// TIA Portal V19 export
FUNCTION_BLOCK "Decoiler_FB"   // FB72, LAD
TITLE = DECOILER MOUNTED ON A ROTATION SYSTEM FOR ON-LINE/OFF-LINE EXCHANGE
// stored: MemoryReserve 100, SetENOAutomatically false
   VAR_INPUT
      AreaInterface : "AreaInterface";
      ZSI : "udt_ZoneSafetyInterface";
      DSI : Struct
         Feed : "udt_DeviceSafetyInterface";
         Jaws : "udt_DeviceSafetyInterface";
         Coupling : "udt_DeviceSafetyInterface";
         SnubberLift : "udt_DeviceSafetyInterface";
         SnubberRoll : "udt_DeviceSafetyInterface";
      END_STRUCT;
      Drive : "TAx_DriveInterface";
      HW_ID_TEL1 : HW_SUBMODULE;
      DataIn : Struct
         DiameterSensor : Int;
         LsPosizioneRazza : Bool;
         Feed : "SpeedMachine_DataIn";
         Jaws : "ValveMachine_DataIn";
         Coupling : "ValveMachine_DataIn";
         SnubberLift : "ValveMachine_DataIn";
         SnubberRoll : "ValveMachine_DataIn";
         Loop : Struct
            Connector : Bool;
            S_MinHigh : Bool;
            S_SpeedAsjust : Bool;
            S_MaxLow : Bool;
         END_STRUCT;
         PneumaticBrake : Struct
            PbOpenClose : Bool;
            PbPartialOpenClose : Bool;
         END_STRUCT;
      END_STRUCT;
      CIn : Struct
         Manager : "Decoiler_Manager";
         PressureRunning : Bool;
      END_STRUCT;
      Config : Struct
         Loop : Struct
            Exist_S_MinHigh : Bool;
            Exist_S_SpeedAdjust : Bool;
         END_STRUCT;
         Feed : "SpeedMachine_Config";
         Jaws : "ValveMachine_Config";
         Coupling : "ValveMachine_Config";
         SnubberLift : "ValveMachine_Config";
         SnubberRoll : "ValveMachine_Config";
         Enable_End_Of_Coil_Using_Loop : Bool := FALSE;
      END_STRUCT;
   END_VAR
   VAR_OUTPUT
      MachineInterface : "MachineInterface";
      DataOut : Struct
         Feed : "SpeedMachine_DataOut";
         Jaws : "ValveMachine_DataOut";
         Coupling : "ValveMachine_DataOut";
         SnubberLift : "ValveMachine_DataOut";
         SnubberRoll : "ValveMachine_DataOut";
         PneumaticBrake : Struct
            V_Open : Bool;
            V_PartialHigh : Bool;
            V_PartialLow : Bool;
            Lp_PbPartialBrake : Bool;
         END_STRUCT;
      END_STRUCT;
      COut : "Decoiler_Status";
   END_VAR
   VAR_IN_OUT
      PersistentValues : "Decoiler_Pers";
   END_VAR
   VAR
      Alarm : Struct
         Feed : "SpeedMachine_Alr";
         Jaws : "ValveAlr";
         Coupling : "ValveAlr";
         SnubberLift : "ValveAlr";
         SnubberRoll : "ValveAlr";
         DimeterSensor : Struct
            SensorrPresetNeed { ExternalAccessible := 'False'; ExternalVisible := 'False'; ExternalWritable := 'False'} : Bool;
         END_STRUCT;
         Loop : Struct
            ConnectorUnplugged : Bool;
         END_STRUCT;
      END_STRUCT;
      Warning : Struct
         EndCoilDetect : Bool;
         Feed : "SpeedMachine_Wng";
         Jaws : "ValveMachine_Wng";
         Coupling { S7_SetPoint := 'True'} : "ValveMachine_Wng";
         SnubberLift { S7_SetPoint := 'True'} : "ValveMachine_Wng";
         SnubberRoll { S7_SetPoint := 'True'} : "ValveMachine_Wng";
         Loop : Struct
            MinHigh : Bool;
         END_STRUCT;
      END_STRUCT;
      HMI : Struct
         Diameter_ButtonPreset : Bool;
         Diameter_PresetValue : Real;
      END_STRUCT;
      Sts : Struct
         StopPosizioneRazza : Bool;
      END_STRUCT;
      Ctrl : Struct
         Jaws : Struct
            AutoOpen : Bool;
            TON_Pause : IEC_TIMER;
            TON_Duration : IEC_TIMER;
         END_STRUCT;
         Brake : Struct
            Open_ReqByMotor : Bool;
            TON_PartialOFF : IEC_TIMER;
            TON_OpenOFF : IEC_TIMER;
         END_STRUCT;
      END_STRUCT;
      DiameterSensor { S7_SetPoint := 'True'} : "Decoiler_DiameterSensor_FB";
      Loop { S7_SetPoint := 'True'} : "Decoiler_Loop_FB";
      Feed { S7_SetPoint := 'True'} : "SpeedMachine_FB";
      PneumaticBrake { S7_SetPoint := 'True'} : "Decoiler_PneumaticBrake";
      Jaws { S7_SetPoint := 'True'} : "ValveMachine_FB";
      SnubberLift { S7_SetPoint := 'True'} : "ValveMachine_FB";
      SnubberRoll { S7_SetPoint := 'True'} : "ValveMachine_FB";
      Coupling { S7_SetPoint := 'True'} : "ValveMachine_FB";
      TON_EndCoilDetect : IEC_TIMER;
      AuxPE : Struct
         LsPosizioneRazza : Bool;
      END_STRUCT;
   END_VAR
   VAR_TEMP
      PE : Struct
         LsPosizioneRazza : Bool;
      END_STRUCT;
      Req : Bool;
   END_VAR
   VAR CONSTANT
      PI : LReal := 3.14159265358979;
   END_VAR
   VAR_TEMP   // added for the SCL form of the ladder/FBD networks
      _w1 : Bool;
   END_VAR
BEGIN

REGION Network 1: <<< MATERIAL FEEDING - PAY-OFF BKW / FWD >>>
END_REGION

REGION Network 2: < Coil Diameter >
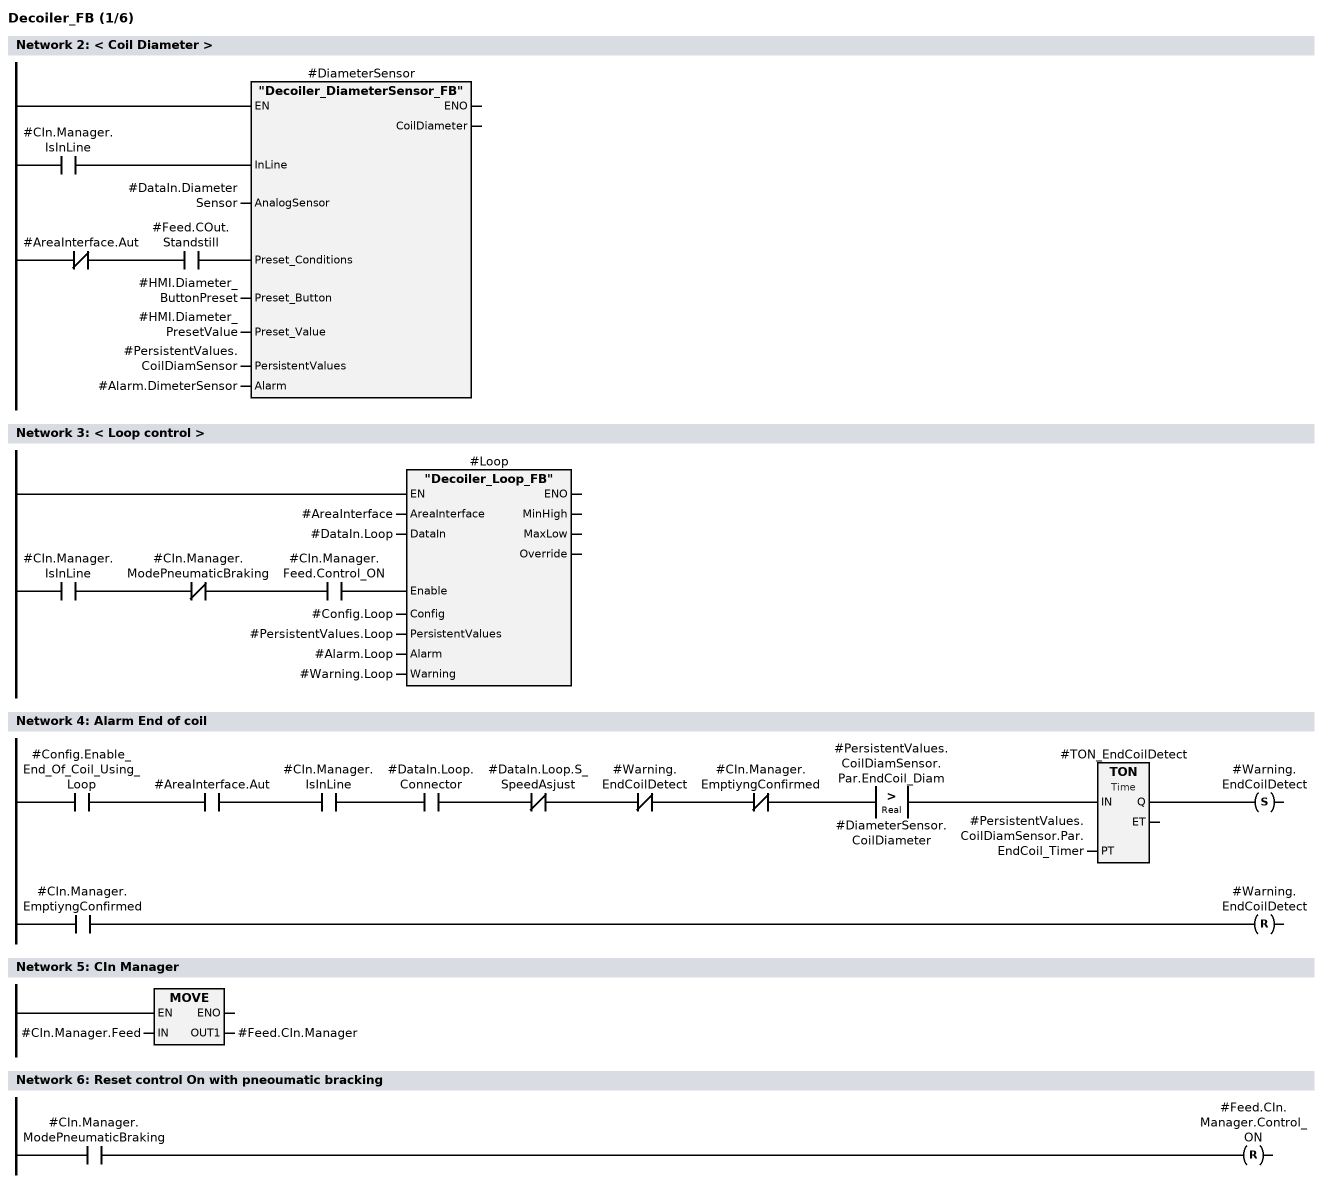
   RUNG wire#powerrail
      #DiameterSensor(InLine := wire#w1, Preset_Conditions := wire#w2, AnalogSensor := #DataIn.DiameterSensor, Preset_Button := #HMI.Diameter_ButtonPreset, Preset_Value := #HMI.Diameter_PresetValue, PersistentValues := #PersistentValues.CoilDiamSensor, Alarm := #Alarm.DimeterSensor, CoilDiameter =>)
   END_RUNG
   RUNG wire#powerrail
      Contact( #CIn.Manager.IsInLine )
   END_RUNG wire#w1
   RUNG wire#powerrail
      I_Contact( #AreaInterface.Aut )
      Contact( #Feed.COut.Standstill )
   END_RUNG wire#w2
   // the same network as SCL:
   #DiameterSensor(InLine := #CIn.Manager.IsInLine,   // "Decoiler_DiameterSensor_FB"
                   AnalogSensor := #DataIn.DiameterSensor,
                   Preset_Conditions := NOT #AreaInterface.Aut AND #Feed.COut.Standstill,
                   Preset_Button := #HMI.Diameter_ButtonPreset,
                   Preset_Value := #HMI.Diameter_PresetValue,
                   PersistentValues := #PersistentValues.CoilDiamSensor,
                   Alarm := #Alarm.DimeterSensor);
END_REGION

REGION Network 3: < Loop control >
   RUNG wire#powerrail
      #Loop(Enable := wire#w1, AreaInterface := #AreaInterface, DataIn := #DataIn.Loop, Config := #Config.Loop, PersistentValues := #PersistentValues.Loop, Alarm := #Alarm.Loop, Warning := #Warning.Loop, MinHigh =>, MaxLow =>, Override =>)
   END_RUNG
   RUNG wire#powerrail
      Contact( #CIn.Manager.IsInLine )
      I_Contact( #CIn.Manager.ModePneumaticBraking )
      Contact( #CIn.Manager.Feed.Control_ON )
   END_RUNG wire#w1
   // the same network as SCL:
   #Loop(AreaInterface := #AreaInterface,   // "Decoiler_Loop_FB"
         DataIn := #DataIn.Loop,
         Enable := #CIn.Manager.IsInLine AND NOT #CIn.Manager.ModePneumaticBraking AND #CIn.Manager.Feed.Control_ON,
         Config := #Config.Loop,
         PersistentValues := #PersistentValues.Loop,
         Alarm := #Alarm.Loop,
         Warning := #Warning.Loop);
END_REGION

REGION Network 4: Alarm End of coil
   RUNG wire#powerrail
      Contact( #Config.Enable_End_Of_Coil_Using_Loop )
      Contact( #AreaInterface.Aut )
      Contact( #CIn.Manager.IsInLine )
      Contact( #DataIn.Loop.Connector )
      I_Contact( #DataIn.Loop.S_SpeedAsjust )
      I_Contact( #Warning.EndCoilDetect )
      I_Contact( #CIn.Manager.EmptiyngConfirmed )
      { S7_Templates := "SrcType := Real" } GT_Contact(in1 := #PersistentValues.CoilDiamSensor.Par.EndCoil_Diam, in2 := #DiameterSensor.CoilDiameter)
      { S7_Templates := "time_type := Time" } #TON_EndCoilDetect.TON(pt := #PersistentValues.CoilDiamSensor.Par.EndCoil_Timer, et =>)
      S_Coil( #Warning.EndCoilDetect )
   END_RUNG
   RUNG wire#powerrail
      Contact( #CIn.Manager.EmptiyngConfirmed )
      R_Coil( #Warning.EndCoilDetect )
   END_RUNG
   // the same network as SCL:
   #TON_EndCoilDetect.TON(IN := #Config.Enable_End_Of_Coil_Using_Loop AND #AreaInterface.Aut AND #CIn.Manager.IsInLine AND #DataIn.Loop.Connector AND NOT #DataIn.Loop.S_SpeedAsjust AND NOT #Warning.EndCoilDetect AND NOT #CIn.Manager.EmptiyngConfirmed AND (#PersistentValues.CoilDiamSensor.Par.EndCoil_Diam > #DiameterSensor.CoilDiameter),
                          PT := #PersistentValues.CoilDiamSensor.Par.EndCoil_Timer);
   IF #TON_EndCoilDetect.Q THEN #Warning.EndCoilDetect := TRUE; END_IF;
   IF #CIn.Manager.EmptiyngConfirmed THEN #Warning.EndCoilDetect := FALSE; END_IF;
END_REGION

REGION Network 5: CIn Manager
   RUNG wire#powerrail
      Move(in := #CIn.Manager.Feed, out1 => #Feed.CIn.Manager)
   END_RUNG
   // the same network as SCL:
   #Feed.CIn.Manager := #CIn.Manager.Feed;
END_REGION

REGION Network 6: Reset control On with pneoumatic bracking
   RUNG wire#powerrail
      Contact( #CIn.Manager.ModePneumaticBraking )
      R_Coil( #Feed.CIn.Manager.Control_ON )
   END_RUNG
   // the same network as SCL:
   IF #CIn.Manager.ModePneumaticBraking THEN #Feed.CIn.Manager.Control_ON := FALSE; END_IF;
END_REGION

REGION Network 7 (SCL): Velocity override with no coupling

   IF NOT #PersistentValues.Coupling.Engaged OR
       NOT #Coupling.COut.Work
   THEN
       #Feed.CIn.Manager.Vel := #PersistentValues.Feed.Man.VelFwdHigh;
   END_IF;
END_REGION

REGION Network 8: CIn Velocity Override
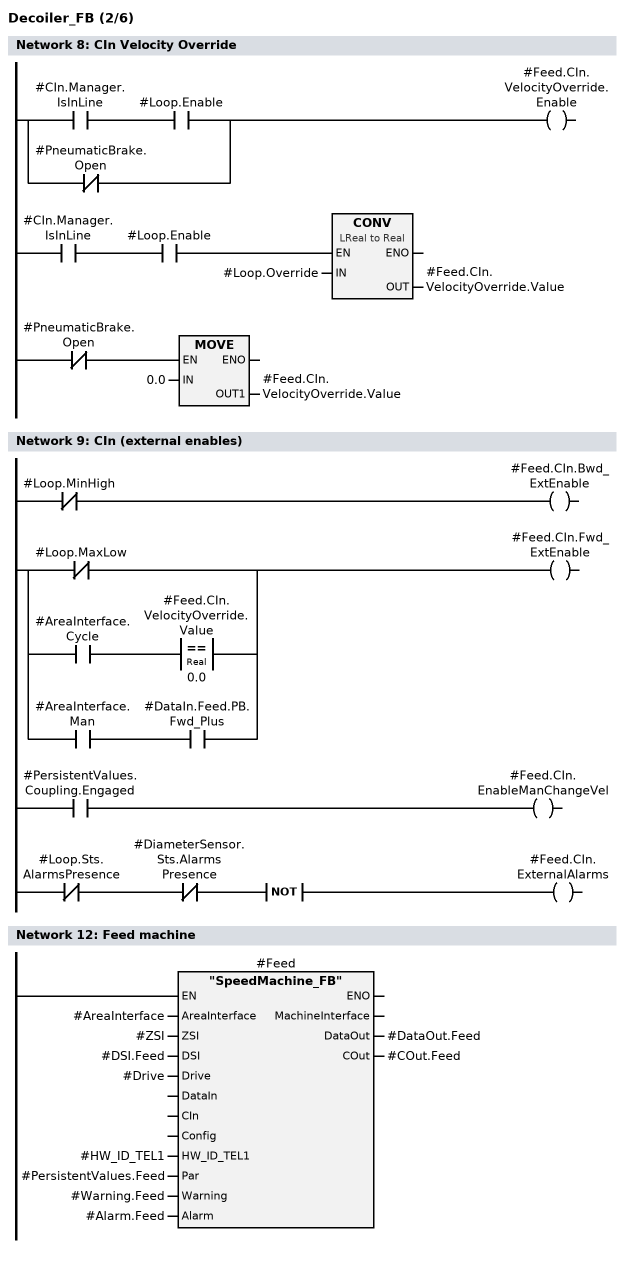
   RUNG wire#powerrail
      Contact( #CIn.Manager.IsInLine )
      Contact( #Loop.Enable )
      wire#w1
      Coil( #Feed.CIn.VelocityOverride.Enable )
   END_RUNG
   RUNG wire#powerrail
      I_Contact( #PneumaticBrake.Open )
   END_RUNG wire#w1
   RUNG wire#powerrail
      Contact( #CIn.Manager.IsInLine )
      Contact( #Loop.Enable )
      { S7_Templates := "[SrcType := LReal, DestType := Real]" } Convert(in := #Loop.Override, out => #Feed.CIn.VelocityOverride.Value)
   END_RUNG
   RUNG wire#powerrail
      I_Contact( #PneumaticBrake.Open )
      Move(in := 0.0, out1 => #Feed.CIn.VelocityOverride.Value)
   END_RUNG
   // the same network as SCL:
   #Feed.CIn.VelocityOverride.Enable := (#CIn.Manager.IsInLine AND #Loop.Enable) OR NOT #PneumaticBrake.Open;
   IF #CIn.Manager.IsInLine AND #Loop.Enable THEN
       #Feed.CIn.VelocityOverride.Value := LREAL_TO_REAL(#Loop.Override);
   END_IF;
   IF NOT #PneumaticBrake.Open THEN #Feed.CIn.VelocityOverride.Value := 0.0; END_IF;
END_REGION

REGION Network 9: CIn (external enables)
   RUNG wire#powerrail
      I_Contact( #Loop.MinHigh )
      Coil( #Feed.CIn.Bwd_ExtEnable )
   END_RUNG
   RUNG wire#powerrail
      I_Contact( #Loop.MaxLow )
      wire#w1
      Coil( #Feed.CIn.Fwd_ExtEnable )
   END_RUNG
   RUNG wire#powerrail
      Contact( #AreaInterface.Cycle )
      { S7_Templates := "SrcType := Real" } EQ_Contact(in1 := #Feed.CIn.VelocityOverride.Value, in2 := 0.0)
   END_RUNG wire#w1
   RUNG wire#powerrail
      Contact( #AreaInterface.Man )
      Contact( #DataIn.Feed.PB.Fwd_Plus )
   END_RUNG wire#w1
   RUNG wire#powerrail
      Contact( #PersistentValues.Coupling.Engaged )
      Coil( #Feed.CIn.EnableManChangeVel )
   END_RUNG
   RUNG wire#powerrail
      I_Contact( #Loop.Sts.AlarmsPresence )
      I_Contact( #DiameterSensor.Sts.AlarmsPresence )
      Not()
      Coil( #Feed.CIn.ExternalAlarms )
   END_RUNG
   // the same network as SCL:
   #Feed.CIn.Bwd_ExtEnable := NOT #Loop.MinHigh;
   #Feed.CIn.Fwd_ExtEnable := NOT #Loop.MaxLow OR (#AreaInterface.Cycle AND (#Feed.CIn.VelocityOverride.Value = 0.0)) OR (#AreaInterface.Man AND #DataIn.Feed.PB.Fwd_Plus);
   #Feed.CIn.EnableManChangeVel := #PersistentValues.Coupling.Engaged;
   #Feed.CIn.ExternalAlarms := NOT (NOT #Loop.Sts.AlarmsPresence AND NOT #DiameterSensor.Sts.AlarmsPresence);
END_REGION

REGION Network 10 (SCL): Config
   #Feed.Config := #Config.Feed;


   #Feed.Config.Ax.LeadScrewPitchVal := #PI * #DiameterSensor.CoilDiameter;
END_REGION

REGION Network 11 (SCL): Data In
   #Feed.DataIn := #DataIn.Feed;

   #PE.LsPosizioneRazza := #DataIn.LsPosizioneRazza AND NOT #AuxPE.LsPosizioneRazza;
   #AuxPE.LsPosizioneRazza := #DataIn.LsPosizioneRazza;

   IF (#DataIn.Feed.PB.Fwd_Plus OR #DataIn.Feed.PB.Bwd_Minus) AND
       #PE.LsPosizioneRazza
   THEN
       #Sts.StopPosizioneRazza := TRUE;
   ELSIF NOT #DataIn.Feed.PB.Fwd_Plus AND
       NOT #DataIn.Feed.PB.Bwd_Minus
   THEN
       #Sts.StopPosizioneRazza := FALSE;
   END_IF;

   #Feed.DataIn.PB.Fwd_Plus := #DataIn.Feed.PB.Fwd_Plus AND NOT #Sts.StopPosizioneRazza;
   #Feed.DataIn.PB.Bwd_Minus := #DataIn.Feed.PB.Bwd_Minus AND NOT #Sts.StopPosizioneRazza;
END_REGION

REGION Network 12: Feed machine
   RUNG wire#powerrail
      #Feed(AreaInterface := #AreaInterface, ZSI := #ZSI, DSI := #DSI.Feed, Drive := #Drive, DataIn :=, CIn :=, Config :=, HW_ID_TEL1 := #HW_ID_TEL1, Par := #PersistentValues.Feed, Warning := #Warning.Feed, Alarm := #Alarm.Feed, MachineInterface =>, DataOut => #DataOut.Feed, COut => #COut.Feed)
   END_RUNG
   // the same network as SCL:
   #Feed(AreaInterface := #AreaInterface,   // "SpeedMachine_FB"
         ZSI := #ZSI,
         DSI := #DSI.Feed,
         Drive := #Drive,
         HW_ID_TEL1 := #HW_ID_TEL1,
         Par := #PersistentValues.Feed,
         Warning := #Warning.Feed,
         Alarm := #Alarm.Feed,
         DataOut => #DataOut.Feed,
         COut => #COut.Feed);
END_REGION

REGION Network 13: < Pneumatic brake >
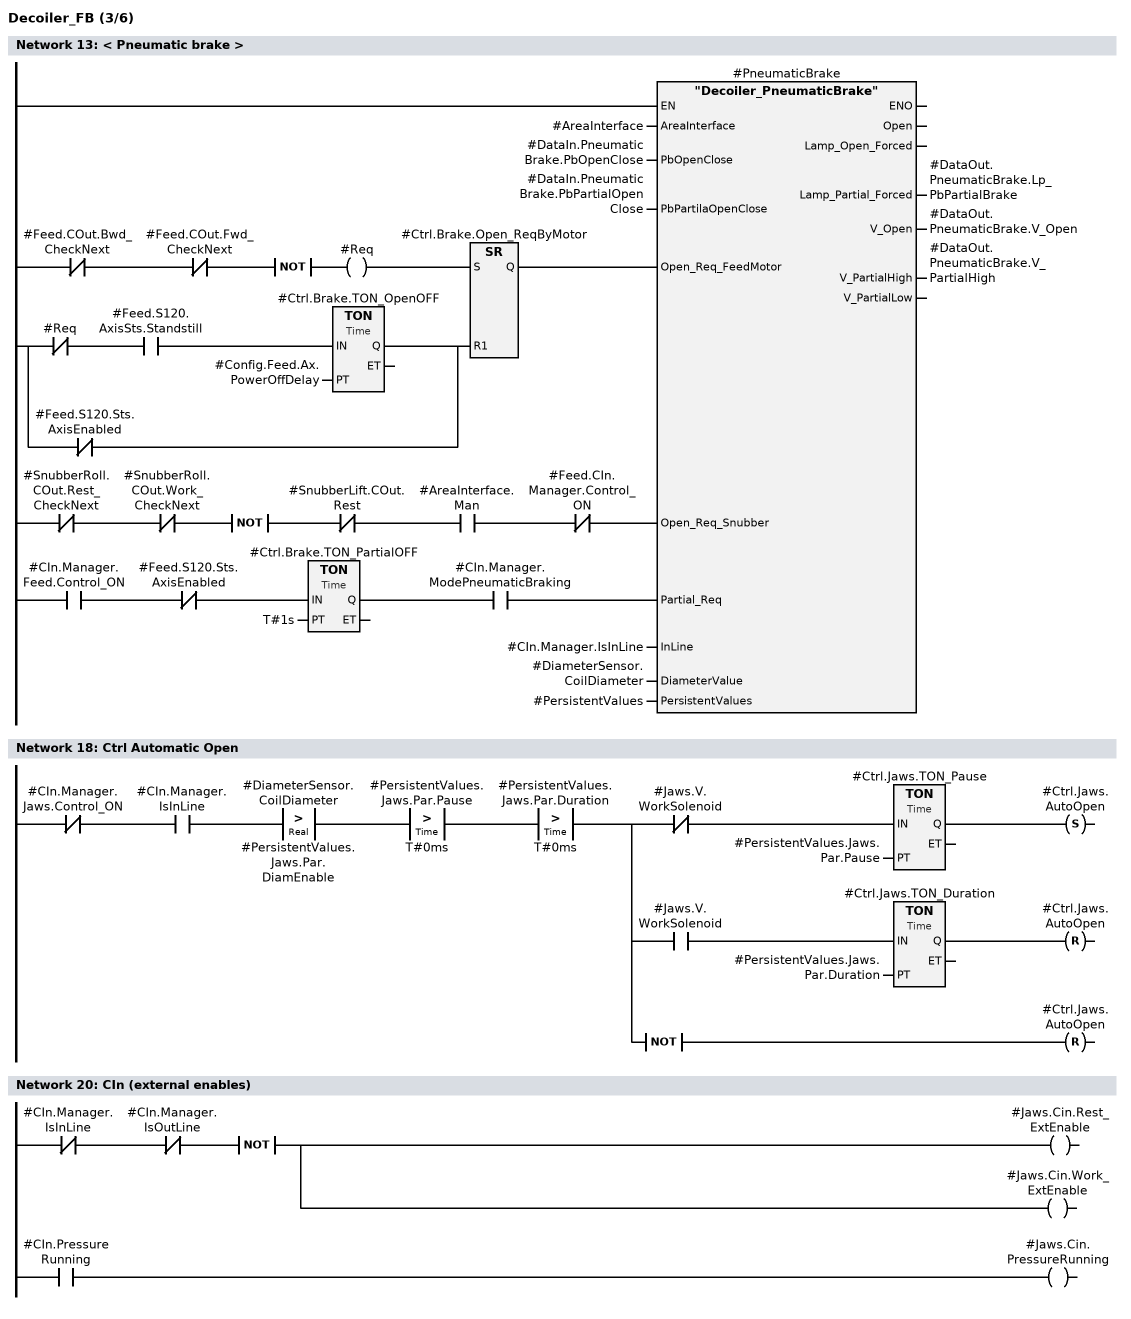
   RUNG wire#powerrail
      #PneumaticBrake(Open_Req_FeedMotor := wire#w2, Open_Req_Snubber := wire#w3, Partial_Req := wire#w4, AreaInterface := #AreaInterface, PbOpenClose := #DataIn.PneumaticBrake.PbOpenClose, PbPartilaOpenClose := #DataIn.PneumaticBrake.PbPartialOpenClose, InLine := #CIn.Manager.IsInLine, DiameterValue := #DiameterSensor.CoilDiameter, PersistentValues := #PersistentValues, Open =>, Lamp_Open_Forced =>, Lamp_Partial_Forced => #DataOut.PneumaticBrake.Lp_PbPartialBrake, V_Open => #DataOut.PneumaticBrake.V_Open, V_PartialHigh => #DataOut.PneumaticBrake.V_PartialHigh, V_PartialLow =>)
   END_RUNG
   RUNG wire#powerrail
      I_Contact( #Feed.COut.Bwd_CheckNext )
      I_Contact( #Feed.COut.Fwd_CheckNext )
      Not()
      Coil( #Req )
      S_SR(operand := #Ctrl.Brake.Open_ReqByMotor, r1 := wire#w1)
   END_RUNG wire#w2
   RUNG wire#powerrail
      I_Contact( #Req )
      Contact( #Feed.S120.AxisSts.Standstill )
      { S7_Templates := "time_type := Time" } #Ctrl.Brake.TON_OpenOFF.TON(pt := #Config.Feed.Ax.PowerOffDelay, et =>)
   END_RUNG wire#w1
   RUNG wire#powerrail
      I_Contact( #Feed.S120.Sts.AxisEnabled )
   END_RUNG wire#w1
   RUNG wire#powerrail
      I_Contact( #SnubberRoll.COut.Rest_CheckNext )
      I_Contact( #SnubberRoll.COut.Work_CheckNext )
      Not()
      I_Contact( #SnubberLift.COut.Rest )
      Contact( #AreaInterface.Man )
      I_Contact( #Feed.CIn.Manager.Control_ON )
   END_RUNG wire#w3
   RUNG wire#powerrail
      Contact( #CIn.Manager.Feed.Control_ON )
      I_Contact( #Feed.S120.Sts.AxisEnabled )
      { S7_Templates := "time_type := Time" } #Ctrl.Brake.TON_PartialOFF.TON(pt := T#1s, et =>)
      Contact( #CIn.Manager.ModePneumaticBraking )
   END_RUNG wire#w4
   // the same network as SCL:
   #Req := NOT (NOT #Feed.COut.Bwd_CheckNext AND NOT #Feed.COut.Fwd_CheckNext);
   #Ctrl.Brake.TON_OpenOFF.TON(IN := NOT #Req AND #Feed.S120.AxisSts.Standstill,
                           PT := #Config.Feed.Ax.PowerOffDelay);
   IF #Req THEN
       #Ctrl.Brake.Open_ReqByMotor := TRUE;   // SR flip-flop
   END_IF;
   IF #Ctrl.Brake.TON_OpenOFF.Q OR NOT #Feed.S120.Sts.AxisEnabled THEN
       #Ctrl.Brake.Open_ReqByMotor := FALSE;
   END_IF;
   #Ctrl.Brake.TON_PartialOFF.TON(IN := #CIn.Manager.Feed.Control_ON AND NOT #Feed.S120.Sts.AxisEnabled,
                           PT := T#1s);
   #PneumaticBrake(AreaInterface := #AreaInterface,   // "Decoiler_PneumaticBrake"
                   PbOpenClose := #DataIn.PneumaticBrake.PbOpenClose,
                   PbPartilaOpenClose := #DataIn.PneumaticBrake.PbPartialOpenClose,
                   Open_Req_FeedMotor := #Ctrl.Brake.Open_ReqByMotor,
                   Open_Req_Snubber := NOT (NOT #SnubberRoll.COut.Rest_CheckNext AND NOT #SnubberRoll.COut.Work_CheckNext) AND NOT #SnubberLift.COut.Rest AND #AreaInterface.Man AND NOT #Feed.CIn.Manager.Control_ON,
                   Partial_Req := #Ctrl.Brake.TON_PartialOFF.Q AND #CIn.Manager.ModePneumaticBraking,
                   InLine := #CIn.Manager.IsInLine,
                   DiameterValue := #DiameterSensor.CoilDiameter,
                   PersistentValues := #PersistentValues,
                   Lamp_Partial_Forced => #DataOut.PneumaticBrake.Lp_PbPartialBrake,
                   V_Open => #DataOut.PneumaticBrake.V_Open,
                   V_PartialHigh => #DataOut.PneumaticBrake.V_PartialHigh);
END_REGION

REGION Network 14: >
END_REGION

REGION Network 15: >
END_REGION

REGION Network 16: >
END_REGION

REGION Network 17: <<< JAWS CLOSE / OPEN >>>
END_REGION

REGION Network 18: Ctrl Automatic Open
   RUNG wire#powerrail
      I_Contact( #CIn.Manager.Jaws.Control_ON )
      Contact( #CIn.Manager.IsInLine )
      { S7_Templates := "SrcType := Real" } GT_Contact(in1 := #DiameterSensor.CoilDiameter, in2 := #PersistentValues.Jaws.Par.DiamEnable)
      { S7_Templates := "SrcType := Time" } GT_Contact(in1 := #PersistentValues.Jaws.Par.Pause, in2 := T#0ms)
      { S7_Templates := "SrcType := Time" } GT_Contact(in1 := #PersistentValues.Jaws.Par.Duration, in2 := T#0ms)
      wire#w1
      I_Contact( #Jaws.V.WorkSolenoid )
      { S7_Templates := "time_type := Time" } #Ctrl.Jaws.TON_Pause.TON(pt := #PersistentValues.Jaws.Par.Pause, et =>)
      S_Coil( #Ctrl.Jaws.AutoOpen )
   END_RUNG
   RUNG wire#w1
      Contact( #Jaws.V.WorkSolenoid )
      { S7_Templates := "time_type := Time" } #Ctrl.Jaws.TON_Duration.TON(pt := #PersistentValues.Jaws.Par.Duration, et =>)
      R_Coil( #Ctrl.Jaws.AutoOpen )
   END_RUNG
   RUNG wire#w1
      Not()
      R_Coil( #Ctrl.Jaws.AutoOpen )
   END_RUNG
   // the same network as SCL:
   #_w1 := NOT #CIn.Manager.Jaws.Control_ON AND #CIn.Manager.IsInLine AND (#DiameterSensor.CoilDiameter > #PersistentValues.Jaws.Par.DiamEnable) AND (#PersistentValues.Jaws.Par.Pause > T#0ms) AND (#PersistentValues.Jaws.Par.Duration > T#0ms);
   #Ctrl.Jaws.TON_Pause.TON(IN := #_w1 AND NOT #Jaws.V.WorkSolenoid, PT := #PersistentValues.Jaws.Par.Pause);
   IF #Ctrl.Jaws.TON_Pause.Q THEN #Ctrl.Jaws.AutoOpen := TRUE; END_IF;
   #Ctrl.Jaws.TON_Duration.TON(IN := #_w1 AND #Jaws.V.WorkSolenoid, PT := #PersistentValues.Jaws.Par.Duration);
   IF #Ctrl.Jaws.TON_Duration.Q THEN #Ctrl.Jaws.AutoOpen := FALSE; END_IF;
   IF NOT #_w1 THEN #Ctrl.Jaws.AutoOpen := FALSE; END_IF;
END_REGION

REGION Network 19 (SCL): CIn Manager
   #Jaws.Cin.Manager := #CIn.Manager.Jaws;

   IF NOT #CIn.Manager.Jaws.Control_ON AND #CIn.Manager.IsInLine THEN

       #Jaws.Cin.Manager.Control_ON := #Ctrl.Jaws.AutoOpen;
       #Jaws.Cin.Manager.Work := #Ctrl.Jaws.AutoOpen;
       #Jaws.Cin.Manager.Rest := FALSE;

   END_IF;
END_REGION

REGION Network 20: CIn (external enables)
   RUNG wire#powerrail
      I_Contact( #CIn.Manager.IsInLine )
      I_Contact( #CIn.Manager.IsOutLine )
      Not()
      wire#w1
      Coil( #Jaws.Cin.Rest_ExtEnable )
   END_RUNG
   RUNG wire#w1
      Coil( #Jaws.Cin.Work_ExtEnable )
   END_RUNG
   RUNG wire#powerrail
      Contact( #CIn.PressureRunning )
      Coil( #Jaws.Cin.PressureRunning )
   END_RUNG
   // the same network as SCL:
   #Jaws.Cin.Rest_ExtEnable := NOT (NOT #CIn.Manager.IsInLine AND NOT #CIn.Manager.IsOutLine);
   #Jaws.Cin.Work_ExtEnable := #Jaws.Cin.Rest_ExtEnable;
   #Jaws.Cin.PressureRunning := #CIn.PressureRunning;
END_REGION

REGION Network 21: Valve machine
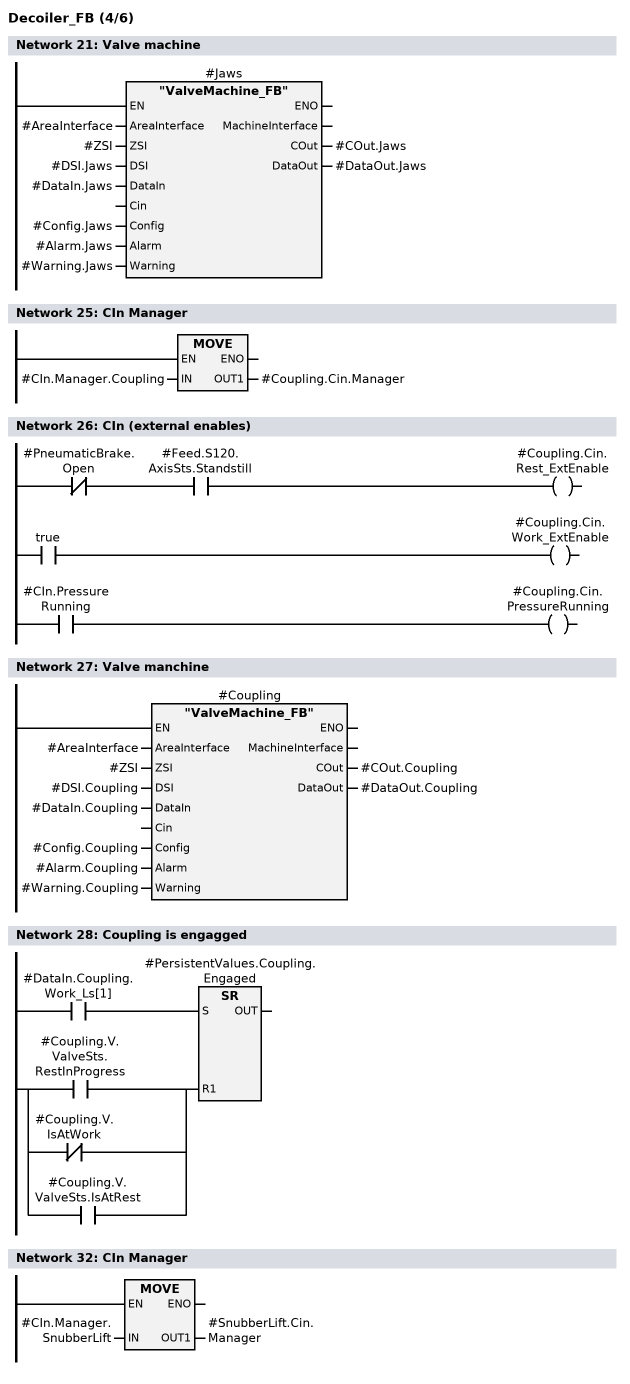
   RUNG wire#powerrail
      #Jaws(AreaInterface := #AreaInterface, ZSI := #ZSI, DSI := #DSI.Jaws, DataIn := #DataIn.Jaws, Cin :=, Config := #Config.Jaws, Alarm := #Alarm.Jaws, Warning := #Warning.Jaws, MachineInterface =>, COut => #COut.Jaws, DataOut => #DataOut.Jaws)
   END_RUNG
   // the same network as SCL:
   #Jaws(AreaInterface := #AreaInterface,   // "ValveMachine_FB"
         ZSI := #ZSI,
         DSI := #DSI.Jaws,
         DataIn := #DataIn.Jaws,
         Config := #Config.Jaws,
         Alarm := #Alarm.Jaws,
         Warning := #Warning.Jaws,
         COut => #COut.Jaws,
         DataOut => #DataOut.Jaws);
END_REGION

REGION Network 22: >
END_REGION

REGION Network 23: >
END_REGION

REGION Network 24: <<< MOTOR COUPLING WORK / REST >>>
END_REGION

REGION Network 25: CIn Manager
   RUNG wire#powerrail
      Move(in := #CIn.Manager.Coupling, out1 => #Coupling.Cin.Manager)
   END_RUNG
   // the same network as SCL:
   #Coupling.Cin.Manager := #CIn.Manager.Coupling;
END_REGION

REGION Network 26: CIn (external enables)
   RUNG wire#powerrail
      I_Contact( #PneumaticBrake.Open )
      Contact( #Feed.S120.AxisSts.Standstill )
      Coil( #Coupling.Cin.Rest_ExtEnable )
   END_RUNG
   RUNG wire#powerrail
      Contact( true )
      Coil( #Coupling.Cin.Work_ExtEnable )
   END_RUNG
   RUNG wire#powerrail
      Contact( #CIn.PressureRunning )
      Coil( #Coupling.Cin.PressureRunning )
   END_RUNG
   // the same network as SCL:
   #Coupling.Cin.Rest_ExtEnable := NOT #PneumaticBrake.Open AND #Feed.S120.AxisSts.Standstill;
   #Coupling.Cin.Work_ExtEnable := true;
   #Coupling.Cin.PressureRunning := #CIn.PressureRunning;
END_REGION

REGION Network 27: Valve manchine
   RUNG wire#powerrail
      #Coupling(AreaInterface := #AreaInterface, ZSI := #ZSI, DSI := #DSI.Coupling, DataIn := #DataIn.Coupling, Cin :=, Config := #Config.Coupling, Alarm := #Alarm.Coupling, Warning := #Warning.Coupling, MachineInterface =>, COut => #COut.Coupling, DataOut => #DataOut.Coupling)
   END_RUNG
   // the same network as SCL:
   #Coupling(AreaInterface := #AreaInterface,   // "ValveMachine_FB"
             ZSI := #ZSI,
             DSI := #DSI.Coupling,
             DataIn := #DataIn.Coupling,
             Config := #Config.Coupling,
             Alarm := #Alarm.Coupling,
             Warning := #Warning.Coupling,
             COut => #COut.Coupling,
             DataOut => #DataOut.Coupling);
END_REGION

REGION Network 28: Coupling is engagged
   RUNG wire#powerrail
      Contact( #DataIn.Coupling.Work_Ls[1] )
      S_SR(operand := #PersistentValues.Coupling.Engaged, r1 := wire#w1)
   END_RUNG
   RUNG wire#powerrail
      Contact( #Coupling.V.ValveSts.RestInProgress )
   END_RUNG wire#w1
   RUNG wire#powerrail
      I_Contact( #Coupling.V.IsAtWork )
   END_RUNG wire#w1
   RUNG wire#powerrail
      Contact( #Coupling.V.ValveSts.IsAtRest )
   END_RUNG wire#w1
   // the same network as SCL:
   IF #DataIn.Coupling.Work_Ls[1] THEN
       #PersistentValues.Coupling.Engaged := TRUE;   // SR flip-flop
   END_IF;
   IF #Coupling.V.ValveSts.RestInProgress OR NOT #Coupling.V.IsAtWork OR #Coupling.V.ValveSts.IsAtRest THEN
       #PersistentValues.Coupling.Engaged := FALSE;
   END_IF;
END_REGION

REGION Network 29: >
END_REGION

REGION Network 30: >
END_REGION

REGION Network 31: <<< SNUBBER LIFT (REST = UP / WORK = DOWN)>>>
END_REGION

REGION Network 32: CIn Manager
   RUNG wire#powerrail
      Move(in := #CIn.Manager.SnubberLift, out1 => #SnubberLift.Cin.Manager)
   END_RUNG
   // the same network as SCL:
   #SnubberLift.Cin.Manager := #CIn.Manager.SnubberLift;
END_REGION

REGION Network 33: CIn (external enables)
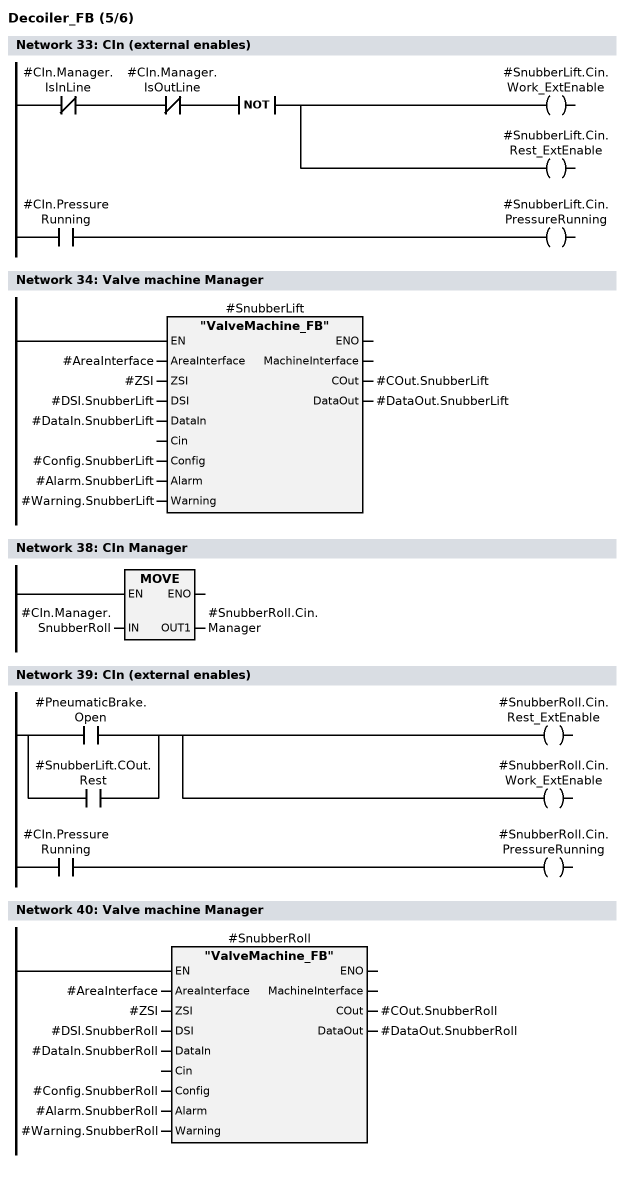
   RUNG wire#powerrail
      I_Contact( #CIn.Manager.IsInLine )
      I_Contact( #CIn.Manager.IsOutLine )
      Not()
      wire#w1
      Coil( #SnubberLift.Cin.Work_ExtEnable )
   END_RUNG
   RUNG wire#w1
      Coil( #SnubberLift.Cin.Rest_ExtEnable )
   END_RUNG
   RUNG wire#powerrail
      Contact( #CIn.PressureRunning )
      Coil( #SnubberLift.Cin.PressureRunning )
   END_RUNG
   // the same network as SCL:
   #SnubberLift.Cin.Work_ExtEnable := NOT (NOT #CIn.Manager.IsInLine AND NOT #CIn.Manager.IsOutLine);
   #SnubberLift.Cin.Rest_ExtEnable := #SnubberLift.Cin.Work_ExtEnable;
   #SnubberLift.Cin.PressureRunning := #CIn.PressureRunning;
END_REGION

REGION Network 34: Valve machine Manager
   RUNG wire#powerrail
      #SnubberLift(AreaInterface := #AreaInterface, ZSI := #ZSI, DSI := #DSI.SnubberLift, DataIn := #DataIn.SnubberLift, Cin :=, Config := #Config.SnubberLift, Alarm := #Alarm.SnubberLift, Warning := #Warning.SnubberLift, MachineInterface =>, COut => #COut.SnubberLift, DataOut => #DataOut.SnubberLift)
   END_RUNG
   // the same network as SCL:
   #SnubberLift(AreaInterface := #AreaInterface,   // "ValveMachine_FB"
                ZSI := #ZSI,
                DSI := #DSI.SnubberLift,
                DataIn := #DataIn.SnubberLift,
                Config := #Config.SnubberLift,
                Alarm := #Alarm.SnubberLift,
                Warning := #Warning.SnubberLift,
                COut => #COut.SnubberLift,
                DataOut => #DataOut.SnubberLift);
END_REGION

REGION Network 35: >
END_REGION

REGION Network 36: >
END_REGION

REGION Network 37: <<< SNUBBER ROLL (REST = BWD / WORK = FWD) >>>
END_REGION

REGION Network 38: CIn Manager
   RUNG wire#powerrail
      Move(in := #CIn.Manager.SnubberRoll, out1 => #SnubberRoll.Cin.Manager)
   END_RUNG
   // the same network as SCL:
   #SnubberRoll.Cin.Manager := #CIn.Manager.SnubberRoll;
END_REGION

REGION Network 39: CIn (external enables)
   RUNG wire#powerrail
      Contact( #PneumaticBrake.Open )
      wire#w1
      Coil( #SnubberRoll.Cin.Rest_ExtEnable )
   END_RUNG
   RUNG wire#powerrail
      Contact( #SnubberLift.COut.Rest )
   END_RUNG wire#w1
   RUNG wire#w1
      Coil( #SnubberRoll.Cin.Work_ExtEnable )
   END_RUNG
   RUNG wire#powerrail
      Contact( #CIn.PressureRunning )
      Coil( #SnubberRoll.Cin.PressureRunning )
   END_RUNG
   // the same network as SCL:
   #SnubberRoll.Cin.Rest_ExtEnable := #PneumaticBrake.Open OR #SnubberLift.COut.Rest;
   #SnubberRoll.Cin.Work_ExtEnable := #SnubberRoll.Cin.Rest_ExtEnable;
   #SnubberRoll.Cin.PressureRunning := #CIn.PressureRunning;
END_REGION

REGION Network 40: Valve machine Manager
   RUNG wire#powerrail
      #SnubberRoll(AreaInterface := #AreaInterface, ZSI := #ZSI, DSI := #DSI.SnubberRoll, DataIn := #DataIn.SnubberRoll, Cin :=, Config := #Config.SnubberRoll, Alarm := #Alarm.SnubberRoll, Warning := #Warning.SnubberRoll, MachineInterface =>, COut => #COut.SnubberRoll, DataOut => #DataOut.SnubberRoll)
   END_RUNG
   // the same network as SCL:
   #SnubberRoll(AreaInterface := #AreaInterface,   // "ValveMachine_FB"
                ZSI := #ZSI,
                DSI := #DSI.SnubberRoll,
                DataIn := #DataIn.SnubberRoll,
                Config := #Config.SnubberRoll,
                Alarm := #Alarm.SnubberRoll,
                Warning := #Warning.SnubberRoll,
                COut => #COut.SnubberRoll,
                DataOut => #DataOut.SnubberRoll);
END_REGION

REGION Network 41: >
END_REGION

REGION Network 42: >
END_REGION

REGION Network 43: <<< MACHINE STATUS >>>
END_REGION

REGION Network 44: COut machine
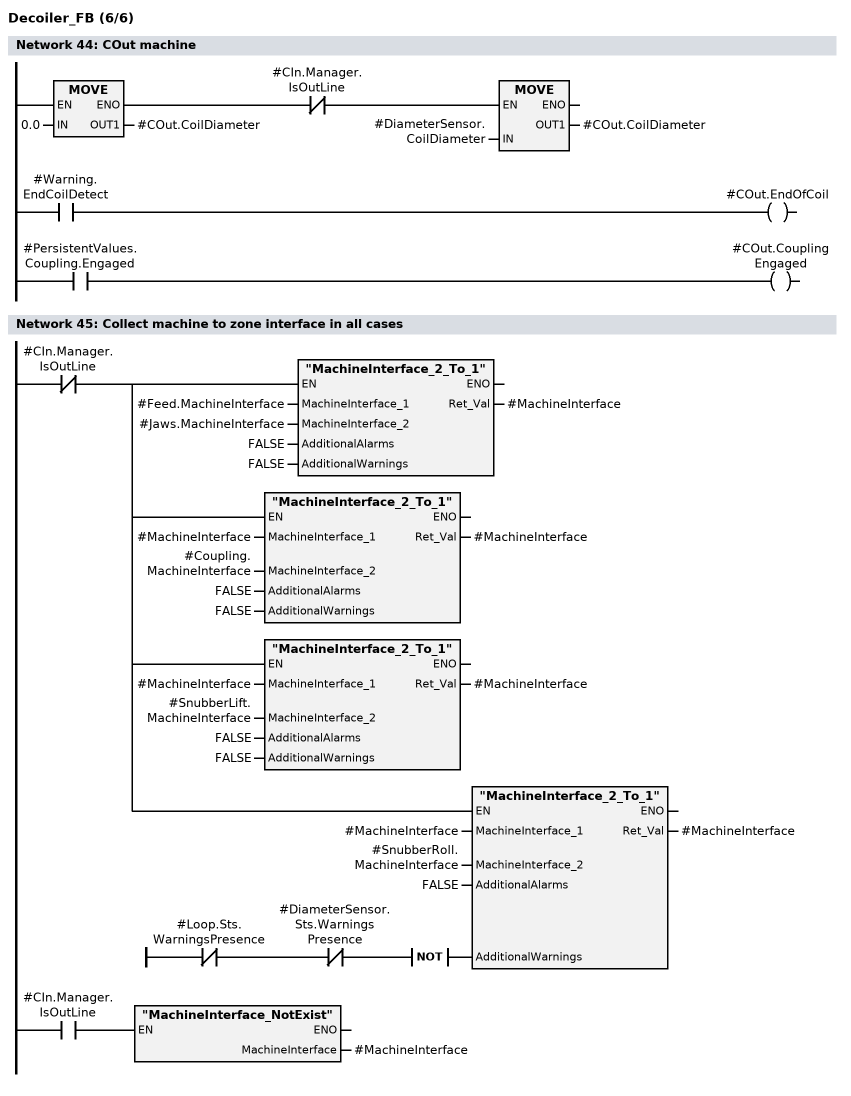
   RUNG wire#powerrail
      Move(in := 0.0, out1 => #COut.CoilDiameter)
      I_Contact( #CIn.Manager.IsOutLine )
      Move(in := #DiameterSensor.CoilDiameter, out1 => #COut.CoilDiameter)
   END_RUNG
   RUNG wire#powerrail
      Contact( #Warning.EndCoilDetect )
      Coil( #COut.EndOfCoil )
   END_RUNG
   RUNG wire#powerrail
      Contact( #PersistentValues.Coupling.Engaged )
      Coil( #COut.CouplingEngaged )
   END_RUNG
   // the same network as SCL:
   #COut.CoilDiameter := 0.0;
   IF NOT #CIn.Manager.IsOutLine THEN #COut.CoilDiameter := #DiameterSensor.CoilDiameter; END_IF;
   #COut.EndOfCoil := #Warning.EndCoilDetect;
   #COut.CouplingEngaged := #PersistentValues.Coupling.Engaged;
END_REGION

REGION Network 45: Collect machine to zone interface in all cases
   RUNG wire#powerrail
      I_Contact( #CIn.Manager.IsOutLine )
      wire#w1
      "MachineInterface_2_To_1"(MachineInterface_1 := #Feed.MachineInterface, MachineInterface_2 := #Jaws.MachineInterface, AdditionalAlarms := FALSE, AdditionalWarnings := FALSE, Ret_Val => #MachineInterface)
   END_RUNG
   RUNG wire#w1
      "MachineInterface_2_To_1"(MachineInterface_1 := #MachineInterface, MachineInterface_2 := #Coupling.MachineInterface, AdditionalAlarms := FALSE, AdditionalWarnings := FALSE, Ret_Val => #MachineInterface)
   END_RUNG
   RUNG wire#w1
      "MachineInterface_2_To_1"(MachineInterface_1 := #MachineInterface, MachineInterface_2 := #SnubberLift.MachineInterface, AdditionalAlarms := FALSE, AdditionalWarnings := FALSE, Ret_Val => #MachineInterface)
   END_RUNG
   RUNG wire#w1
      "MachineInterface_2_To_1"(AdditionalWarnings := wire#w2, MachineInterface_1 := #MachineInterface, MachineInterface_2 := #SnubberRoll.MachineInterface, AdditionalAlarms := FALSE, Ret_Val => #MachineInterface)
   END_RUNG
   RUNG wire#powerrail
      I_Contact( #Loop.Sts.WarningsPresence )
      I_Contact( #DiameterSensor.Sts.WarningsPresence )
      Not()
   END_RUNG wire#w2
   RUNG wire#powerrail
      Contact( #CIn.Manager.IsOutLine )
      "MachineInterface_NotExist"(MachineInterface => #MachineInterface)
   END_RUNG
   // the same network as SCL:
   IF NOT #CIn.Manager.IsOutLine THEN
       #MachineInterface := "MachineInterface_2_To_1"(MachineInterface_1 := #Feed.MachineInterface,
                               MachineInterface_2 := #Jaws.MachineInterface,
                               AdditionalAlarms := FALSE,
                               AdditionalWarnings := FALSE);
       #MachineInterface := "MachineInterface_2_To_1"(MachineInterface_1 := #MachineInterface,
                               MachineInterface_2 := #Coupling.MachineInterface,
                               AdditionalAlarms := FALSE,
                               AdditionalWarnings := FALSE);
       #MachineInterface := "MachineInterface_2_To_1"(MachineInterface_1 := #MachineInterface,
                               MachineInterface_2 := #SnubberLift.MachineInterface,
                               AdditionalAlarms := FALSE,
                               AdditionalWarnings := FALSE);
       #MachineInterface := "MachineInterface_2_To_1"(MachineInterface_1 := #MachineInterface,
                               MachineInterface_2 := #SnubberRoll.MachineInterface,
                               AdditionalAlarms := FALSE,
                               AdditionalWarnings := NOT (NOT #Loop.Sts.WarningsPresence AND NOT #DiameterSensor.Sts.WarningsPresence));
   END_IF;
   IF #CIn.Manager.IsOutLine THEN "MachineInterface_NotExist"(MachineInterface => #MachineInterface); END_IF;
END_REGION

REGION Network 46: >
END_REGION

REGION Network 47: >
END_REGION

REGION Network 48: >
END_REGION
END_FUNCTION_BLOCK
